ABB RobotStudio station: tuto1.rsstn

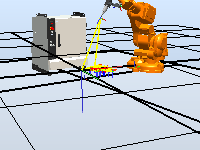
Station tuto1 (saved by RobotStudio format 3)
Controller Sistema1, task T_ROB1: task frame (RAPID world) sits at (1500, 0, 400) mm in the station
Controller Sistema1
  mechanical unit ROB_1: IRB140_5_81__01, 6 joints, base frame (0, 0, 0) mm
Layout (positions relative to the parent item):
  - IRB140_5_81__01 [mechanism, from Robots\IRB140_5_81__01.rslib] at (1500, 0, 400) mm; joint values [-1.2609, 0.3579, -0.6855, 2.4225, -0.9972, -2.6268] (rad or m)
  - IRC5_Singel-Cabinet [part, from Equipment\IRC5_Singel-Cabinet.rslib] at (-626.3, -13.51, 100) mm, rotated rx 90 ry 0 rz 90.54 deg
  - MyTool [mechanism, from Training Objects\myTool.rslib] at (1649.51, -584.8, 1183.88) mm, rotated rx -152.62 ry 61.49 rz 100.62 deg
Attachment: MyTool is attached to IRB140_5_81__01 / Link6
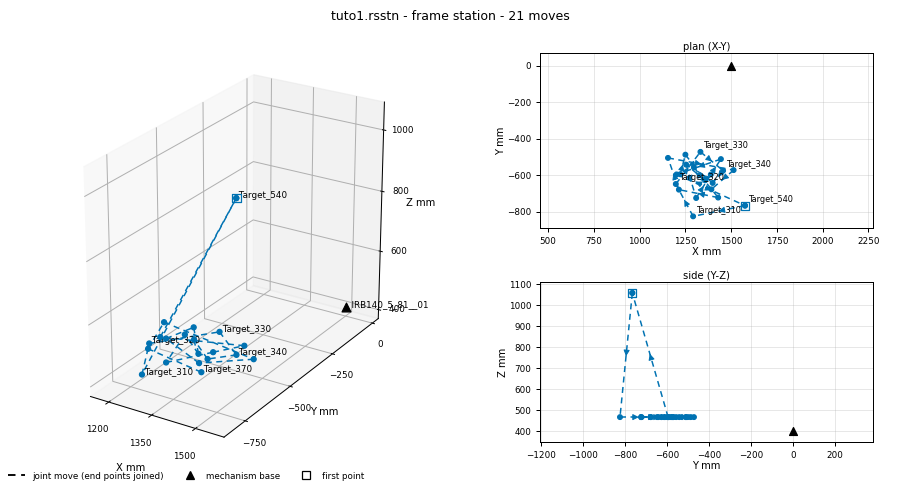
[picture p0: tool path of tuto1.rsstn in frame station, 21 of 21 moves have a stored position in this frame; points joined in program order, loops and branches not executed]
Targets, tools, work objects and paths stored in the station, written as RAPID:
! task T_ROB1
MODULE CalibData
  PERS tooldata MyTool:=[TRUE,[[31.792631019,0,229.638935148],[0.945518576,0,0.325568154,0]],[1,[0,0,1],[1,0,0,0],0,0,0]];
  TASK PERS wobjdata Workobject_1:=[FALSE,TRUE,"",[[0,-241.738827836,67.0901308],[1,0,0,0]],[[0,0,0],[1,0,0,0]]];
ENDMODULE

! task T_ROB1
MODULE Module1
  CONST robtarget Target_310:=[[-207.652832031,-582.438964844,0],[0,0.766044443,0.64278761,0],[-1,1,-2,1],[9E9,9E9,9E9,9E9,9E9,9E9]];
  CONST robtarget Target_320:=[[-302.208007813,-405.773681641,0],[0,0.766044443,0.64278761,0],[0,-2,-1,6],[9E9,9E9,9E9,9E9,9E9,9E9]];
  CONST robtarget Target_330:=[[-167.640380859,-230.099853516,0],[0,0.766044443,0.64278761,0],[-2,-2,-3,1],[9E9,9E9,9E9,9E9,9E9,9E9]];
  CONST robtarget Target_340:=[[-43.809326172,-332.403320313,0],[0,0.766044443,0.64278761,0],[-2,-1,-4,1],[9E9,9E9,9E9,9E9,9E9,9E9]];
  CONST robtarget Target_350:=[[-100.91015625,-399.837158203,0],[0,0.766044443,0.64278761,0],[-2,0,-5,1],[9E9,9E9,9E9,9E9,9E9,9E9]];
  CONST robtarget Target_360:=[[-203.477783203,-314.919433594,0],[0,0.766044443,0.64278761,0],[-2,0,-5,1],[9E9,9E9,9E9,9E9,9E9,9E9]];
  CONST robtarget Target_370:=[[-70.813476562,-479.770019531,0],[0,0.766044443,0.64278761,0],[-2,-1,-4,0],[9E9,9E9,9E9,9E9,9E9,9E9]];
  CONST robtarget Target_380:=[[-285.333251953,-436.612548828,0],[0,0.766044443,0.64278761,0],[-2,-2,-3,1],[9E9,9E9,9E9,9E9,9E9,9E9]];
  CONST robtarget Target_390:=[[-345.013183594,-263.082275391,0],[0,0.766044443,0.64278761,0],[-2,-2,-3,1],[9E9,9E9,9E9,9E9,9E9,9E9]];
  CONST robtarget Target_420:=[[13.627441406,-329.596435547,0],[0,0.766044443,0.64278761,0],[-2,-1,-4,1],[9E9,9E9,9E9,9E9,9E9,9E9]];
  CONST robtarget Target_430:=[[-107.833251953,-434.733398438,0],[0,0.766044443,0.64278761,0],[-1,0,-5,1],[9E9,9E9,9E9,9E9,9E9,9E9]];
  CONST robtarget Target_440:=[[-278.184814453,-352.316162109,0],[0,0.766044443,0.64278761,0],[-2,0,-5,1],[9E9,9E9,9E9,9E9,9E9,9E9]];
  CONST robtarget Target_450:=[[-249.843017578,-245.385253906,0],[0,0.766044443,0.64278761,0],[-2,-1,-4,1],[9E9,9E9,9E9,9E9,9E9,9E9]];
  CONST robtarget Target_480:=[[-141.9765625,-385.512451172,0],[0,0.766044443,0.64278761,0],[-2,-1,-4,1],[9E9,9E9,9E9,9E9,9E9,9E9]];
  CONST robtarget Target_490:=[[-245.778076172,-299.910888672,0],[0,0.766044443,0.64278761,0],[-2,-1,-4,1],[9E9,9E9,9E9,9E9,9E9,9E9]];
  CONST robtarget Target_500:=[[-191.046142578,-482.264892578,0],[0,0.766044443,0.64278761,0],[-2,-1,-4,1],[9E9,9E9,9E9,9E9,9E9,9E9]];
  CONST robtarget Target_510:=[[-111.029296875,-354.013671875,0],[0,0.766044443,0.64278761,0],[-2,-2,-3,1],[9E9,9E9,9E9,9E9,9E9,9E9]];
  CONST robtarget Target_520:=[[-55.799804687,-269.524169922,0],[0,0.766044443,0.64278761,0],[-2,-1,-4,1],[9E9,9E9,9E9,9E9,9E9,9E9]];
  CONST robtarget Target_530:=[[-298.242675781,-353.310791016,0],[0,0.766044443,0.64278761,0],[-2,0,-5,1],[9E9,9E9,9E9,9E9,9E9,9E9]];
  CONST robtarget Target_540:=[[75.939761559,-765.473990699,658.616288324],[0.0545479,0.746483111,0.616649789,-0.243988789],[-1,1,-2,1],[9E9,9E9,9E9,9E9,9E9,9E9]];
  PROC Path_10()
    MoveJ Target_540,v1000,z200,MyTool\WObj:=wobj0;
    MoveJ Target_310,v1000,z200,MyTool\WObj:=Workobject_1;
    MoveJ Target_320,v1000,z200,MyTool\WObj:=Workobject_1;
    MoveJ Target_330,v1000,z200,MyTool\WObj:=Workobject_1;
    MoveJ Target_340,v1000,z200,MyTool\WObj:=Workobject_1;
    MoveJ Target_350,v1000,z200,MyTool\WObj:=Workobject_1;
    MoveJ Target_360,v1000,z200,MyTool\WObj:=Workobject_1;
    MoveJ Target_370,v1000,z200,MyTool\WObj:=Workobject_1;
    MoveJ Target_380,v1000,z200,MyTool\WObj:=Workobject_1;
    MoveJ Target_390,v1000,z200,MyTool\WObj:=Workobject_1;
    MoveJ Target_420,v1000,z200,MyTool\WObj:=Workobject_1;
    MoveJ Target_430,v1000,z200,MyTool\WObj:=Workobject_1;
    MoveJ Target_440,v1000,z200,MyTool\WObj:=Workobject_1;
    MoveJ Target_450,v1000,z200,MyTool\WObj:=Workobject_1;
    MoveJ Target_480,v1000,z200,MyTool\WObj:=Workobject_1;
    MoveJ Target_490,v1000,z200,MyTool\WObj:=Workobject_1;
    MoveJ Target_500,v1000,z200,MyTool\WObj:=Workobject_1;
    MoveJ Target_510,v1000,z200,MyTool\WObj:=Workobject_1;
    MoveJ Target_520,v1000,z200,MyTool\WObj:=Workobject_1;
    MoveJ Target_530,v1000,z200,MyTool\WObj:=Workobject_1;
    MoveJ Target_540,v1000,z200,MyTool\WObj:=wobj0;
  ENDPROC
ENDMODULE

